// TIA Portal V20 export
FUNCTION_BLOCK "FB_ReadDateAndTime"   // FB46, SCL
{ S7_Optimized_Access := 'TRUE' }
// stored: MemoryReserve 100, SetENOAutomatically false
   VAR
      sDateAndTime : DTL;
      sCurrentDT : Struct
         sYear : UInt;
         sMonth : USInt;
         sDay : USInt;
         sHour : USInt;
         sMinute : USInt;
         sSecond : USInt;
         sNanoSecond : UDInt;
      END_STRUCT;
   END_VAR
   VAR_TEMP
      tRetVal : Int;
   END_VAR
BEGIN
   REGION Description header 
       //==================================================================================
       // POSALUX Swiss SA / (C) Copyright 2025
       //----------------------------------------------------------------------------------
       // Title: FB_ReadDateAndTime
       // Comment/Function: Reading the date and time of the PLC
       // Author: Fabien WALDT
       // Engineering: TIA Portal v20
       //----------------------------------------------------------------------------------
       // Change log table:
       // Version  | Date     | Expert in charge | Changes applied
       // ---------|----------|------------------|-----------------------------------------
       // 00.00.01 | 20251017 | WFA              | First released version
       // =================================================================================
   END_REGION

   REGION Lecture Date et Heure
       #tRetVal :=RD_SYS_T(OUT => #sDateAndTime);
       #sCurrentDT.sYear       := #sDateAndTime.YEAR;
       #sCurrentDT.sMonth      := #sDateAndTime.MONTH;
       #sCurrentDT.sHour      := #sDateAndTime.HOUR;
       #sCurrentDT.sMinute     := #sDateAndTime.MINUTE;
       #sCurrentDT.sSecond     := #sDateAndTime.SECOND;
       #sCurrentDT.sNanoSecond := #sDateAndTime.NANOSECOND;
   END_REGION
END_FUNCTION_BLOCK
